FUNCTION ThetaM3 : REAL
VAR_INPUT
END_VAR
VAR
END_VAR

END_FUNCTION

(* stored: Version 1.1.0.1, ProductVersion 3.1.4024.6
   POU ThetaM3: Id {0fae6683-3e5e-42fb-97db-8e03e9fa75ff}, SpecialFunc None *)
